TYPE ST_Robot_Mitsubishi_Packet_1103 :
STRUCT
	// Packet number - 1103. 8B This is separated due to the need of on trigger confirmation.
	// From robot.
	// Robot Dependency confirmed.
	// Trigger.
	
	Header							: DINT := 1103;													// Packet header.
	
	DepencencyState					: DINT;
END_STRUCT
END_TYPE

(* stored: Version 1.1.0.1, ProductVersion 3.1.4024.3
   DUT ST_Robot_Mitsubishi_Packet_1103: Id {d5d35ac4-e3b3-4932-b05a-81597605e9a7} *)
